{attribute addProperty BoxType "KL6211"}
{attribute addProperty Id "StatusAT %I*UINT000Parameter_InAT %I*UDINT000ASI_In_Slave_1_StatusAT %I*USINT000ASI_In_Slave_3_Slave_2AT %I*USINT000ASI_In_Slave_5_Slave_4AT %I*USINT000ASI_In_Slave_7_Slave_6AT %I*USINT000ASI_In_Slave_9_Slave_8AT %I*USINT000ASI_In_Slave_11_Slave_10AT %I*USINT000ControlAT %Q*UINT000Parameter_OutAT %Q*UDINT000ASI_Out_Slave_1_ControlAT %Q*USINT000ASI_Out_Slave_3_Slave_2AT %Q*USINT000ASI_Out_Slave_5_Slave_4AT %Q*USINT000ASI_Out_Slave_7_Slave_6AT %Q*USINT000ASI_Out_Slave_9_Slave_8AT %Q*USINT000ASI_Out_Slave_11_Slave_10AT %Q*USINT000"}
{attribute addProperty CRC "2757078489"}
{attribute addProperty SizeInBites "0"}
{attribute addProperty SizeInBytes "0"}
TYPE Channel_A455ADD9 :
STRUCT
	{attribute addProperty Name "Status"}
	Status AT %I* : UINT;
	{attribute addProperty Name "Parameter_In"}
	Parameter_In AT %I* : UDINT;
	{attribute addProperty Name "ASI_In_Slave_1_Status"}
	ASI_In_Slave_1_Status AT %I* : USINT;
	{attribute addProperty Name "ASI_In_Slave_3_Slave_2"}
	ASI_In_Slave_3_Slave_2 AT %I* : USINT;
	{attribute addProperty Name "ASI_In_Slave_5_Slave_4"}
	ASI_In_Slave_5_Slave_4 AT %I* : USINT;
	{attribute addProperty Name "ASI_In_Slave_7_Slave_6"}
	ASI_In_Slave_7_Slave_6 AT %I* : USINT;
	{attribute addProperty Name "ASI_In_Slave_9_Slave_8"}
	ASI_In_Slave_9_Slave_8 AT %I* : USINT;
	{attribute addProperty Name "ASI_In_Slave_11_Slave_10"}
	ASI_In_Slave_11_Slave_10 AT %I* : USINT;
	{attribute addProperty Name "Control"}
	Control AT %Q* : UINT;
	{attribute addProperty Name "Parameter_Out"}
	Parameter_Out AT %Q* : UDINT;
	{attribute addProperty Name "ASI_Out_Slave_1_Control"}
	ASI_Out_Slave_1_Control AT %Q* : USINT;
	{attribute addProperty Name "ASI_Out_Slave_3_Slave_2"}
	ASI_Out_Slave_3_Slave_2 AT %Q* : USINT;
	{attribute addProperty Name "ASI_Out_Slave_5_Slave_4"}
	ASI_Out_Slave_5_Slave_4 AT %Q* : USINT;
	{attribute addProperty Name "ASI_Out_Slave_7_Slave_6"}
	ASI_Out_Slave_7_Slave_6 AT %Q* : USINT;
	{attribute addProperty Name "ASI_Out_Slave_9_Slave_8"}
	ASI_Out_Slave_9_Slave_8 AT %Q* : USINT;
	{attribute addProperty Name "ASI_Out_Slave_11_Slave_10"}
	ASI_Out_Slave_11_Slave_10 AT %Q* : USINT;
END_STRUCT
END_TYPE

(* stored: Version 1.2.0.0, ProductVersion 3.1.4024.9
   DUT Channel_A455ADD9: Id {7e8c1dcb-6560-4a93-b69e-c096ee6ed65a} *)
